Universal Robots PolyScope program: static_blocks.urp

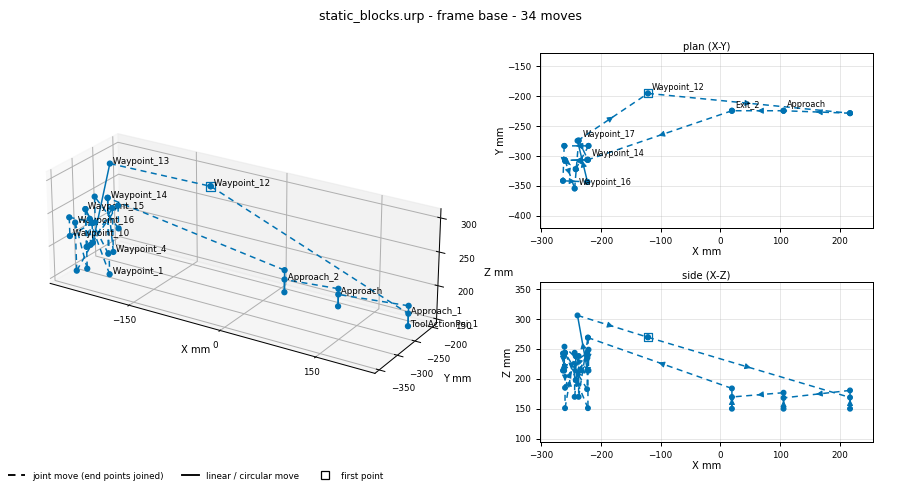
[picture p0: tool path of static_blocks.urp in frame base, 34 of 34 moves have a stored position in this frame; points joined in program order, loops and branches not executed]
Program static_blocks (installation=default directory=/programs/usbdisk createdIn=5.3.1.64192 lastSavedIn=5.3.1.64192 robotSerialNumber=20195300365)
Calibrated DH parameters: a=[-0.000093, -0.190649, -0.212673, 0.000091, -0.000205, 0]; d=[0.151591, 44.061648, -42.488068, -1.442789, 0.085322, 0.091911]; alpha=[1.570082, -0.003447, 0.007513, 1.572293, -1.571904, 0]; deltaTheta=[0, -0.672656, 0.728185, -0.055522, 0.000005, 0]
BeforeStart
  URCap Gripper Activate (Robotiq_Grippers, Robotiq Inc.) dataModel(ResetAndActivateKey=true)
  Wait Sleep waitTime=2
  URCap Gripper (Robotiq_Grippers, Robotiq Inc.) dataModel(position=50.0, force=100.0, speed=100.0, positionInDouble=50.0, forceInDouble=100.0, speedInDouble=100.0, slaveIds=[9], blocking=true)
Robot Program (runOnlyOnce=true)
  MoveJ speed 60 deg/s, acceleration 80 deg/s^2 (useActiveTCP=true) feature=Base
    Waypoint Waypoint_12: TCP in base x=-121.283 y=-195.081 z=269.514 mm, rx=-2.167 ry=2.2415 rz=-0.0076 rad; joints [-88.099, -64.133, -118.46, -88.049, 91.631, -85.899] deg
  next := "large_1"
  Loop Counting (count=11) loopVariable(name=Loop_1)
    'Block selection'
    If next ≟ "large_1"
      URCap Palletizing (pallet-impl, Universal Robots) dataModel(palletFeature=Base, isPalletizing=true, rememberTraversal=false, Length(key=objectHeight value=0.01 unit=M), Variable(key=layerNumberVariable, variable(name=Pallet_1_lno, initializeExpression=1)), Variable(key=layerCountingVariable, variable(name=Pallet_1_lct, initializeExpression=1)), Variable(key=handleSeparatorVariable, variable(name=Pallet_1_sep, initializeExpression=False)), Variable(key=totalCountVariable, variable(name=Pallet_1_tct, initializeExpression=1)), Variable(key=name, variable(name=Large_1)), Variable(key=referencePoint, variable(featureName=referencePoint)), Variable(key=separatorPoint, variable(featureName=separatorPoint)), Variable(key=globalCountingVariable, variable(name=Pallet_1_cnt1, initializeExpression=1))); state(isChildrenLocked=true)
        URCap Patterns (pallet-impl, Universal Robots) state(isChildrenLocked=true)
          URCap Pattern (pallet-impl, Universal Robots) dataModel(UUID=37575b9b-24e8-4b53-bf02-43d1c72f6588, patternType=LINE, objects=4, Variable(key=nameVariable, variable(name=Line_Pattern_1))); state(isChildrenLocked=true)
            URCap Item (pallet-impl, Universal Robots) dataModel(UUID=94ef26eb-0406-42c0-9c7a-a5d3f7661bb4, patternType=LINE, index=0, calibrationDeltaTheta=[3.1764833014445715E-7, -0.6726562497450229, 0.7281850965771859, -0.055521791881094344, 5.417975891638949E-6, -3.308891861480978E-7], calibrationA=[-9.327832644612732E-5, -0.19064944224513533, -0.21267280235524616, 9.135661128094068E-5, -2.046441875520248E-4, 0.0], calibrationD=[0.15159127566255157, 44.06164831948618, -42.48806757161077, -1.4427889341768174, 0.08532194966640622, 0.09191068481194639], calibrationAlpha=[1.5700823634315826, -0.0034467901999681192, 0.007512569451791506, 1.5722928534010268, -1.5719039470931155, 0.0], calibrationJointChecksum=[-1322437199, -1322307948, -1493592214, -1327938167, -1330538947, -1329494862], calibrationStatus=2, calibrationValidChecksum=true, baseToFeature=[0.0, 0.0, 0.0, 0.0, 0.0, 0.0], TCPOffset=[2.6818013665053098E-6, -8.523257610526525E-7, 3.187511623176098E-6, -5.221405753076122E-6, 1.0916503052633558E-5, 1.7823756412515186E-5], JointPositions(key=jointpositions, JointPosition(key=[1], Angle(key=pos value=-0.386285 unit=RAD)), JointPosition(key=[2], Angle(key=pos value=-1.772217 unit=RAD)), JointPosition(key=[3], Angle(key=pos value=-2.142066 unit=RAD)), JointPosition(key=[4], Angle(key=pos value=-0.803353 unit=RAD)), JointPosition(key=[5], Angle(key=pos value=1.570932 unit=RAD)), JointPosition(key=[6], Angle(key=pos value=-0.3815 unit=RAD))), Variable(key=variable, variable(name=StartItem_1)))
            URCap Item (pallet-impl, Universal Robots) dataModel(UUID=a723c821-374d-4fb7-a72e-4b4fba4af77d, patternType=LINE, index=1, calibrationDeltaTheta=[3.1764833014445715E-7, -0.6726562497450229, 0.7281850965771859, -0.055521791881094344, 5.417975891638949E-6, -3.308891861480978E-7], calibrationA=[-9.327832644612732E-5, -0.19064944224513533, -0.21267280235524616, 9.135661128094068E-5, -2.046441875520248E-4, 0.0], calibrationD=[0.15159127566255157, 44.06164831948618, -42.48806757161077, -1.4427889341768174, 0.08532194966640622, 0.09191068481194639], calibrationAlpha=[1.5700823634315826, -0.0034467901999681192, 0.007512569451791506, 1.5722928534010268, -1.5719039470931155, 0.0], calibrationJointChecksum=[-1322437199, -1322307948, -1493592214, -1327938167, -1330538947, -1329494862], calibrationStatus=2, calibrationValidChecksum=true, baseToFeature=[0.0, 0.0, 0.0, 0.0, 0.0, 0.0], TCPOffset=[-4.482752550050151E-6, -1.082257494983141E-5, -1.6687113393309971E-6, -3.080320700071801E-6, 2.847478995674553E-5, -7.719056088527975E-5], JointPositions(key=jointpositions, JointPosition(key=[1], Angle(key=pos value=-0.845813 unit=RAD)), JointPosition(key=[2], Angle(key=pos value=-2.443735 unit=RAD)), JointPosition(key=[3], Angle(key=pos value=-1.007946 unit=RAD)), JointPosition(key=[4], Angle(key=pos value=-1.263676 unit=RAD)), JointPosition(key=[5], Angle(key=pos value=1.569273 unit=RAD)), JointPosition(key=[6], Angle(key=pos value=-0.846194 unit=RAD))), Variable(key=variable, variable(name=EndItem_1)))
        URCap Layers (pallet-impl, Universal Robots) dataModel(separators=[false], selectedPatterns=[37575b9b-24e8-4b53-bf02-43d1c72f6588])
        URCap At Each Item (pallet-impl, Universal Robots) dataModel(selectedPattern=37575b9b-24e8-4b53-bf02-43d1c72f6588, selectedPosition=94ef26eb-0406-42c0-9c7a-a5d3f7661bb4, Approach_calibrationDeltaTheta=[3.1764833014445715E-7, -0.6726562497450229, 0.7281850965771859, -0.055521791881094344, 5.417975891638949E-6, -3.308891861480978E-7], Approach_calibrationA=[-9.327832644612732E-5, -0.19064944224513533, -0.21267280235524616, 9.135661128094068E-5, -2.046441875520248E-4, 0.0], Approach_calibrationD=[0.15159127566255157, 44.06164831948618, -42.48806757161077, -1.4427889341768174, 0.08532194966640622, 0.09191068481194639], Approach_calibrationAlpha=[1.5700823634315826, -0.0034467901999681192, 0.007512569451791506, 1.5722928534010268, -1.5719039470931155, 0.0], Approach_calibrationJointChecksum=[-1322437199, -1322307948, -1493592214, -1327938167, -1330538947, -1329494862], Approach_calibrationStatus=2, Approach_calibrationValidChecksum=true, Approach_baseToFeature=[0.0, 0.0, 0.0, 0.0, 0.0, 0.0], Approach_TCPOffset=[-1.4110221621399521E-6, -9.056105289340088E-6, -4.040316261583188E-6, -7.025378227736759E-6, 4.9770386753854616E-6, -2.713524910439085E-5], Exit_calibrationDeltaTheta=[3.1764833014445715E-7, -0.6726562497450229, 0.7281850965771859, -0.055521791881094344, 5.417975891638949E-6, -3.308891861480978E-7], Exit_calibrationA=[-9.327832644612732E-5, -0.19064944224513533, -0.21267280235524616, 9.135661128094068E-5, -2.046441875520248E-4, 0.0], Exit_calibrationD=[0.15159127566255157, 44.06164831948618, -42.48806757161077, -1.4427889341768174, 0.08532194966640622, 0.09191068481194639], Exit_calibrationAlpha=[1.5700823634315826, -0.0034467901999681192, 0.007512569451791506, 1.5722928534010268, -1.5719039470931155, 0.0], Exit_calibrationJointChecksum=[-1322437199, -1322307948, -1493592214, -1327938167, -1330538947, -1329494862], Exit_calibrationStatus=2, Exit_calibrationValidChecksum=true, Exit_baseToFeature=[0.0, 0.0, 0.0, 0.0, 0.0, 0.0], Exit_TCPOffset=[4.440688230411549E-6, 1.0608106728315914E-5, 6.984684250199713E-6, -3.32523645938351E-5, 8.927854697233474E-6, -3.551786211011088E-5], currentWizardState=LANDING, Pose(key=refBaseToFeature, Position(key=posePosition, Length(key=X value=0 unit=M), Length(key=Y value=0 unit=M), Length(key=Z value=0 unit=M)), Rotation(key=poseRotation, Angle(key=RX value=0 unit=RAD), Angle(key=RY value=0 unit=RAD), Angle(key=RZ value=0 unit=RAD))), Pose(key=refPose, Position(key=posePosition, Length(key=X value=0.216857 unit=M), Length(key=Y value=-0.228211 unit=M), Length(key=Z value=0.149941 unit=M)), Rotation(key=poseRotation, Angle(key=RX value=2.221569 unit=RAD), Angle(key=RY value=-2.213073 unit=RAD), Angle(key=RZ value=-0.006933 unit=RAD))), JointPositions(key=Approach_jointpositions, JointPosition(key=[1], Angle(key=pos value=-0.386188 unit=RAD)), JointPosition(key=[2], Angle(key=pos value=-1.712734 unit=RAD)), JointPosition(key=[3], Angle(key=pos value=-2.099671 unit=RAD)), JointPosition(key=[4], Angle(key=pos value=-0.90523 unit=RAD)), JointPosition(key=[5], Angle(key=pos value=1.571526 unit=RAD)), JointPosition(key=[6], Angle(key=pos value=-0.381836 unit=RAD))), JointPositions(key=Exit_jointpositions, JointPosition(key=[1], Angle(key=pos value=-0.386112 unit=RAD)), JointPosition(key=[2], Angle(key=pos value=-1.679803 unit=RAD)), JointPosition(key=[3], Angle(key=pos value=-2.069692 unit=RAD)), JointPosition(key=[4], Angle(key=pos value=-0.968137 unit=RAD)), JointPosition(key=[5], Angle(key=pos value=1.571865 unit=RAD)), JointPosition(key=[6], Angle(key=pos value=-0.382075 unit=RAD))))
          URCap Generated Movements (pallet-impl, Universal Robots) state(isChildrenLocked=true)
            MoveJ speed 60 deg/s, acceleration 80 deg/s^2 (useActiveTCP=true) feature=referencePoint
              Waypoint Approach_1: TCP in base x=216.866 y=-228.21 z=168.787 mm, rx=2.2216 ry=-2.213 rz=-0.0069 rad; joints [-22.126, -98.133, -120.3, -51.868, 90.041, -21.878] deg; TCP offset x=0 y=0 z=0 mm, rx=0 ry=0 rz=0 rad; feature pose in base x=216.857 y=-228.211 z=149.941 mm, rx=2.2216 ry=-2.2131 rz=-0.0069 rad
            MoveL speed 250 mm/s, acceleration 1200 mm/s^2 (useActiveTCP=true) feature(featureName=referencePoint)
              Waypoint ToolActionPoi_1: TCP in base x=216.857 y=-228.211 z=149.941 mm, rx=2.2216 ry=-2.2131 rz=-0.0069 rad; joints [-22.133, -101.542, -122.731, -46.028, 90.007, -21.858] deg; TCP offset x=0 y=0 z=0 mm, rx=0 ry=0 rz=0 rad
            Folder Tool action
              URCap Gripper (Robotiq_Grippers, Robotiq Inc.) dataModel(position=100.0, force=100.0, speed=100.0, positionInDouble=100.0, forceInDouble=100.0, speedInDouble=100.0, slaveIds=[9], blocking=true)
            MoveL speed 250 mm/s, acceleration 1200 mm/s^2 (useActiveTCP=true) feature(featureName=referencePoint)
              Waypoint Exit_1: motionParameters(blendRadius=0.015); TCP in base x=216.847 y=-228.216 z=180.576 mm, rx=2.2216 ry=-2.213 rz=-0.007 rad; joints [-22.124, -96.246, -118.586, -55.47, 90.06, -21.895] deg; TCP offset x=0 y=0 z=0 mm, rx=0 ry=0 rz=0 rad
    ElseIf next ≟ "small_1"
      URCap Palletizing (pallet-impl, Universal Robots) dataModel(palletFeature=Base, isPalletizing=true, rememberTraversal=false, Length(key=objectHeight value=0.01 unit=M), Variable(key=layerNumberVariable, variable(name=Pallet_1_lno_1, initializeExpression=1)), Variable(key=layerCountingVariable, variable(name=Pallet_1_lct_1, initializeExpression=1)), Variable(key=handleSeparatorVariable, variable(name=Pallet_1_sep_1, initializeExpression=False)), Variable(key=totalCountVariable, variable(name=Pallet_1_tct_1, initializeExpression=1)), Variable(key=name, variable(name=Small_1)), Variable(key=referencePoint, variable(featureName=referencePoin_1)), Variable(key=separatorPoint, variable(featureName=separatorPoin_1)), Variable(key=globalCountingVariable, variable(name=Pallet_1_cnt2, initializeExpression=1))); state(isChildrenLocked=true)
        URCap Patterns (pallet-impl, Universal Robots) state(isChildrenLocked=true)
          URCap Pattern (pallet-impl, Universal Robots) dataModel(UUID=8f5fe08d-2c45-49f2-8f1a-65c607567d74, patternType=LINE, objects=4, Variable(key=nameVariable, variable(name=Line_Pattern_2))); state(isChildrenLocked=true)
            URCap Item (pallet-impl, Universal Robots) dataModel(UUID=ef528854-cb52-475c-81ed-63f5d340cd60, patternType=LINE, index=0, calibrationDeltaTheta=[3.1764833014445715E-7, -0.6726562497450229, 0.7281850965771859, -0.055521791881094344, 5.417975891638949E-6, -3.308891861480978E-7], calibrationA=[-9.327832644612732E-5, -0.19064944224513533, -0.21267280235524616, 9.135661128094068E-5, -2.046441875520248E-4, 0.0], calibrationD=[0.15159127566255157, 44.06164831948618, -42.48806757161077, -1.4427889341768174, 0.08532194966640622, 0.09191068481194639], calibrationAlpha=[1.5700823634315826, -0.0034467901999681192, 0.007512569451791506, 1.5722928534010268, -1.5719039470931155, 0.0], calibrationJointChecksum=[-1322437199, -1322307948, -1493592214, -1327938167, -1330538947, -1329494862], calibrationStatus=2, calibrationValidChecksum=true, baseToFeature=[0.0, 0.0, 0.0, 0.0, 0.0, 0.0], TCPOffset=[7.196090374694819E-7, -7.525119034013095E-7, 2.3613486090923175E-6, -5.861788620822338E-6, -1.7185264349297415E-5, 1.0867011174151283E-5], JointPositions(key=jointpositions, JointPosition(key=[1], Angle(key=pos value=-0.579147 unit=RAD)), JointPosition(key=[2], Angle(key=pos value=-1.475214 unit=RAD)), JointPosition(key=[3], Angle(key=pos value=-2.46543 unit=RAD)), JointPosition(key=[4], Angle(key=pos value=-0.776185 unit=RAD)), JointPosition(key=[5], Angle(key=pos value=1.570404 unit=RAD)), JointPosition(key=[6], Angle(key=pos value=-0.573518 unit=RAD))), Variable(key=variable, variable(name=StartItem_2)))
            URCap Item (pallet-impl, Universal Robots) dataModel(UUID=c15b3bae-27b4-4f22-a9be-ccead8772f48, patternType=LINE, index=1, calibrationDeltaTheta=[3.1764833014445715E-7, -0.6726562497450229, 0.7281850965771859, -0.055521791881094344, 5.417975891638949E-6, -3.308891861480978E-7], calibrationA=[-9.327832644612732E-5, -0.19064944224513533, -0.21267280235524616, 9.135661128094068E-5, -2.046441875520248E-4, 0.0], calibrationD=[0.15159127566255157, 44.06164831948618, -42.48806757161077, -1.4427889341768174, 0.08532194966640622, 0.09191068481194639], calibrationAlpha=[1.5700823634315826, -0.0034467901999681192, 0.007512569451791506, 1.5722928534010268, -1.5719039470931155, 0.0], calibrationJointChecksum=[-1322437199, -1322307948, -1493592214, -1327938167, -1330538947, -1329494862], calibrationStatus=2, calibrationValidChecksum=true, baseToFeature=[0.0, 0.0, 0.0, 0.0, 0.0, 0.0], TCPOffset=[6.867596638648887E-6, 1.6127585317354809E-6, -1.4517486032261662E-5, -5.9295253787075885E-6, 7.61064027945187E-5, -1.3647353319639889E-5], JointPositions(key=jointpositions, JointPosition(key=[1], Angle(key=pos value=-1.056839 unit=RAD)), JointPosition(key=[2], Angle(key=pos value=-2.273802 unit=RAD)), JointPosition(key=[3], Angle(key=pos value=-1.326947 unit=RAD)), JointPosition(key=[4], Angle(key=pos value=-1.113261 unit=RAD)), JointPosition(key=[5], Angle(key=pos value=1.568262 unit=RAD)), JointPosition(key=[6], Angle(key=pos value=-1.055578 unit=RAD))), Variable(key=variable, variable(name=EndItem_2)))
        URCap Layers (pallet-impl, Universal Robots) dataModel(separators=[false], selectedPatterns=[8f5fe08d-2c45-49f2-8f1a-65c607567d74])
        URCap At Each Item (pallet-impl, Universal Robots) dataModel(selectedPattern=8f5fe08d-2c45-49f2-8f1a-65c607567d74, selectedPosition=ef528854-cb52-475c-81ed-63f5d340cd60, Approach_calibrationDeltaTheta=[3.1764833014445715E-7, -0.6726562497450229, 0.7281850965771859, -0.055521791881094344, 5.417975891638949E-6, -3.308891861480978E-7], Approach_calibrationA=[-9.327832644612732E-5, -0.19064944224513533, -0.21267280235524616, 9.135661128094068E-5, -2.046441875520248E-4, 0.0], Approach_calibrationD=[0.15159127566255157, 44.06164831948618, -42.48806757161077, -1.4427889341768174, 0.08532194966640622, 0.09191068481194639], Approach_calibrationAlpha=[1.5700823634315826, -0.0034467901999681192, 0.007512569451791506, 1.5722928534010268, -1.5719039470931155, 0.0], Approach_calibrationJointChecksum=[-1322437199, -1322307948, -1493592214, -1327938167, -1330538947, -1329494862], Approach_calibrationStatus=2, Approach_calibrationValidChecksum=true, Approach_baseToFeature=[0.0, 0.0, 0.0, 0.0, 0.0, 0.0], Approach_TCPOffset=[-1.8296166631182054E-6, -5.2785861738846585E-6, 4.523678061779668E-6, -2.6542376188082585E-5, -8.975232779585173E-6, -3.1784731117598936E-5], Exit_calibrationDeltaTheta=[3.1764833014445715E-7, -0.6726562497450229, 0.7281850965771859, -0.055521791881094344, 5.417975891638949E-6, -3.308891861480978E-7], Exit_calibrationA=[-9.327832644612732E-5, -0.19064944224513533, -0.21267280235524616, 9.135661128094068E-5, -2.046441875520248E-4, 0.0], Exit_calibrationD=[0.15159127566255157, 44.06164831948618, -42.48806757161077, -1.4427889341768174, 0.08532194966640622, 0.09191068481194639], Exit_calibrationAlpha=[1.5700823634315826, -0.0034467901999681192, 0.007512569451791506, 1.5722928534010268, -1.5719039470931155, 0.0], Exit_calibrationJointChecksum=[-1322437199, -1322307948, -1493592214, -1327938167, -1330538947, -1329494862], Exit_calibrationStatus=2, Exit_calibrationValidChecksum=true, Exit_baseToFeature=[0.0, 0.0, 0.0, 0.0, 0.0, 0.0], Exit_TCPOffset=[-1.517237854353759E-6, -9.613929180279923E-6, -6.434422402695761E-6, 9.261849516252882E-6, 1.6687881217173567E-5, -3.51484445230019E-5], currentWizardState=LANDING, Pose(key=refBaseToFeature, Position(key=posePosition, Length(key=X value=0 unit=M), Length(key=Y value=0 unit=M), Length(key=Z value=0 unit=M)), Rotation(key=poseRotation, Angle(key=RX value=0 unit=RAD), Angle(key=RY value=0 unit=RAD), Angle(key=RZ value=0 unit=RAD))), Pose(key=refPose, Position(key=posePosition, Length(key=X value=0.105616 unit=M), Length(key=Y value=-0.224089 unit=M), Length(key=Z value=0.149939 unit=M)), Rotation(key=poseRotation, Angle(key=RX value=2.221562 unit=RAD), Angle(key=RY value=-2.213091 unit=RAD), Angle(key=RZ value=-0.006958 unit=RAD))), JointPositions(key=Approach_jointpositions, JointPosition(key=[1], Angle(key=pos value=-0.578996 unit=RAD)), JointPosition(key=[2], Angle(key=pos value=-1.398829 unit=RAD)), JointPosition(key=[3], Angle(key=pos value=-2.412 unit=RAD)), JointPosition(key=[4], Angle(key=pos value=-0.906009 unit=RAD)), JointPosition(key=[5], Angle(key=pos value=1.571251 unit=RAD)), JointPosition(key=[6], Angle(key=pos value=-0.573984 unit=RAD))), JointPositions(key=Exit_jointpositions, JointPosition(key=[1], Angle(key=pos value=-0.578911 unit=RAD)), JointPosition(key=[2], Angle(key=pos value=-1.367711 unit=RAD)), JointPosition(key=[3], Angle(key=pos value=-2.384276 unit=RAD)), JointPosition(key=[4], Angle(key=pos value=-0.96485 unit=RAD)), JointPosition(key=[5], Angle(key=pos value=1.571588 unit=RAD)), JointPosition(key=[6], Angle(key=pos value=-0.574219 unit=RAD))))
          URCap Generated Movements (pallet-impl, Universal Robots) state(isChildrenLocked=true)
            MoveJ speed 60 deg/s, acceleration 80 deg/s^2 (useActiveTCP=true) feature=referencePoin_1
              Waypoint Approach: TCP in base x=105.622 y=-224.087 z=168.076 mm, rx=2.2216 ry=-2.213 rz=-0.007 rad; joints [-33.173, -80.148, -138.197, -51.911, 90.026, -32.887] deg; TCP offset x=0 y=0 z=0 mm, rx=0 ry=0 rz=0 rad; feature pose in base x=105.616 y=-224.089 z=149.939 mm, rx=2.2216 ry=-2.2131 rz=-0.007 rad
            MoveL speed 250 mm/s, acceleration 1200 mm/s^2 (useActiveTCP=true) feature(featureName=referencePoin_1)
              Waypoint ToolActionPoint: TCP in base x=105.616 y=-224.089 z=149.939 mm, rx=2.2216 ry=-2.2131 rz=-0.007 rad; joints [-33.183, -84.525, -141.258, -44.472, 89.978, -32.86] deg; TCP offset x=0 y=0 z=0 mm, rx=0 ry=0 rz=0 rad
            Folder Tool action
              URCap Gripper (Robotiq_Grippers, Robotiq Inc.) dataModel(position=100.0, force=100.0, speed=100.0, positionInDouble=100.0, forceInDouble=100.0, speedInDouble=100.0, slaveIds=[9], blocking=true)
            MoveL speed 250 mm/s, acceleration 1200 mm/s^2 (useActiveTCP=true) feature(featureName=referencePoin_1)
              Waypoint Exit: motionParameters(blendRadius=0.015); TCP in base x=105.626 y=-224.087 z=176.77 mm, rx=2.2216 ry=-2.213 rz=-0.0069 rad; joints [-33.167, -78.363, -136.608, -55.283, 90.045, -32.9] deg; TCP offset x=0 y=0 z=0 mm, rx=0 ry=0 rz=0 rad
    Else 
      URCap Palletizing (pallet-impl, Universal Robots) dataModel(palletFeature=Base, isPalletizing=true, rememberTraversal=false, Length(key=objectHeight value=0.01 unit=M), Variable(key=layerNumberVariable, variable(name=Pallet_3_lno, initializeExpression=1)), Variable(key=layerCountingVariable, variable(name=Pallet_3_lct, initializeExpression=1)), Variable(key=handleSeparatorVariable, variable(name=Pallet_3_sep, initializeExpression=False)), Variable(key=totalCountVariable, variable(name=Pallet_3_tct, initializeExpression=1)), Variable(key=name, variable(name=Small_2)), Variable(key=referencePoint, variable(featureName=referencePoin_2)), Variable(key=separatorPoint, variable(featureName=separatorPoin_2)), Variable(key=globalCountingVariable, variable(name=Pallet_3_cnt1, initializeExpression=1))); state(isChildrenLocked=true)
        URCap Patterns (pallet-impl, Universal Robots) state(isChildrenLocked=true)
          URCap Pattern (pallet-impl, Universal Robots) dataModel(UUID=574e648a-9869-4bcb-a6fe-864b98b65979, patternType=LINE, objects=4, Variable(key=nameVariable, variable(name=Line_Pattern_3))); state(isChildrenLocked=true)
            URCap Item (pallet-impl, Universal Robots) dataModel(UUID=3619f09d-97e3-4d4e-aeec-a5329e7c8f8b, patternType=LINE, index=0, calibrationDeltaTheta=[3.1764833014445715E-7, -0.6726562497450229, 0.7281850965771859, -0.055521791881094344, 5.417975891638949E-6, -3.308891861480978E-7], calibrationA=[-9.327832644612732E-5, -0.19064944224513533, -0.21267280235524616, 9.135661128094068E-5, -2.046441875520248E-4, 0.0], calibrationD=[0.15159127566255157, 44.06164831948618, -42.48806757161077, -1.4427889341768174, 0.08532194966640622, 0.09191068481194639], calibrationAlpha=[1.5700823634315826, -0.0034467901999681192, 0.007512569451791506, 1.5722928534010268, -1.5719039470931155, 0.0], calibrationJointChecksum=[-1322437199, -1322307948, -1493592214, -1327938167, -1330538947, -1329494862], calibrationStatus=2, calibrationValidChecksum=true, baseToFeature=[0.0, 0.0, 0.0, 0.0, 0.0, 0.0], TCPOffset=[-1.471914889417114E-7, -9.062111944835999E-6, 4.858574105065516E-6, -6.559488045899108E-6, -1.3766923162685491E-5, -5.608483778319356E-6], JointPositions(key=jointpositions, JointPosition(key=[1], Angle(key=pos value=-0.869663 unit=RAD)), JointPosition(key=[2], Angle(key=pos value=-1.338984 unit=RAD)), JointPosition(key=[3], Angle(key=pos value=-2.567281 unit=RAD)), JointPosition(key=[4], Angle(key=pos value=-0.808969 unit=RAD)), JointPosition(key=[5], Angle(key=pos value=1.569596 unit=RAD)), JointPosition(key=[6], Angle(key=pos value=-0.863997 unit=RAD))), Variable(key=variable, variable(name=StartItem_3)))
            URCap Item (pallet-impl, Universal Robots) dataModel(UUID=43353e96-12ed-4b99-95b5-f18523ae2f1f, patternType=LINE, index=1, calibrationDeltaTheta=[3.1764833014445715E-7, -0.6726562497450229, 0.7281850965771859, -0.055521791881094344, 5.417975891638949E-6, -3.308891861480978E-7], calibrationA=[-9.327832644612732E-5, -0.19064944224513533, -0.21267280235524616, 9.135661128094068E-5, -2.046441875520248E-4, 0.0], calibrationD=[0.15159127566255157, 44.06164831948618, -42.48806757161077, -1.4427889341768174, 0.08532194966640622, 0.09191068481194639], calibrationAlpha=[1.5700823634315826, -0.0034467901999681192, 0.007512569451791506, 1.5722928534010268, -1.5719039470931155, 0.0], calibrationJointChecksum=[-1322437199, -1322307948, -1493592214, -1327938167, -1330538947, -1329494862], calibrationStatus=2, calibrationValidChecksum=true, baseToFeature=[0.0, 0.0, 0.0, 0.0, 0.0, 0.0], TCPOffset=[-2.699244438297832E-6, -1.993162529571879E-7, -2.2601341719635792E-5, 2.6517761326188484E-5, 3.333393093251858E-5, 1.450252224784447E-5], JointPositions(key=jointpositions, JointPosition(key=[1], Angle(key=pos value=-1.246701 unit=RAD)), JointPosition(key=[2], Angle(key=pos value=-2.204283 unit=RAD)), JointPosition(key=[3], Angle(key=pos value=-1.452761 unit=RAD)), JointPosition(key=[4], Angle(key=pos value=-1.055644 unit=RAD)), JointPosition(key=[5], Angle(key=pos value=1.567749 unit=RAD)), JointPosition(key=[6], Angle(key=pos value=-1.24482 unit=RAD))), Variable(key=variable, variable(name=EndItem_3)))
        URCap Layers (pallet-impl, Universal Robots) dataModel(separators=[false], selectedPatterns=[574e648a-9869-4bcb-a6fe-864b98b65979])
        URCap At Each Item (pallet-impl, Universal Robots) dataModel(selectedPattern=574e648a-9869-4bcb-a6fe-864b98b65979, selectedPosition=3619f09d-97e3-4d4e-aeec-a5329e7c8f8b, Approach_calibrationDeltaTheta=[3.1764833014445715E-7, -0.6726562497450229, 0.7281850965771859, -0.055521791881094344, 5.417975891638949E-6, -3.308891861480978E-7], Approach_calibrationA=[-9.327832644612732E-5, -0.19064944224513533, -0.21267280235524616, 9.135661128094068E-5, -2.046441875520248E-4, 0.0], Approach_calibrationD=[0.15159127566255157, 44.06164831948618, -42.48806757161077, -1.4427889341768174, 0.08532194966640622, 0.09191068481194639], Approach_calibrationAlpha=[1.5700823634315826, -0.0034467901999681192, 0.007512569451791506, 1.5722928534010268, -1.5719039470931155, 0.0], Approach_calibrationJointChecksum=[-1322437199, -1322307948, -1493592214, -1327938167, -1330538947, -1329494862], Approach_calibrationStatus=2, Approach_calibrationValidChecksum=true, Approach_baseToFeature=[0.0, 0.0, 0.0, 0.0, 0.0, 0.0], Approach_TCPOffset=[1.7216837140676677E-6, -3.506743741481938E-6, -1.0808390142336144E-6, -1.6443935207651089E-6, 4.86080167331034E-6, -2.9982690882012256E-5], Exit_calibrationDeltaTheta=[3.1764833014445715E-7, -0.6726562497450229, 0.7281850965771859, -0.055521791881094344, 5.417975891638949E-6, -3.308891861480978E-7], Exit_calibrationA=[-9.327832644612732E-5, -0.19064944224513533, -0.21267280235524616, 9.135661128094068E-5, -2.046441875520248E-4, 0.0], Exit_calibrationD=[0.15159127566255157, 44.06164831948618, -42.48806757161077, -1.4427889341768174, 0.08532194966640622, 0.09191068481194639], Exit_calibrationAlpha=[1.5700823634315826, -0.0034467901999681192, 0.007512569451791506, 1.5722928534010268, -1.5719039470931155, 0.0], Exit_calibrationJointChecksum=[-1322437199, -1322307948, -1493592214, -1327938167, -1330538947, -1329494862], Exit_calibrationStatus=2, Exit_calibrationValidChecksum=true, Exit_baseToFeature=[0.0, 0.0, 0.0, 0.0, 0.0, 0.0], Exit_TCPOffset=[-4.7682124618142474E-7, -1.929772925179929E-6, -1.986456084873689E-6, 4.125717686270397E-6, -2.831162655691365E-6, 4.997597875419577E-8], currentWizardState=LANDING, Pose(key=refBaseToFeature, Position(key=posePosition, Length(key=X value=0 unit=M), Length(key=Y value=0 unit=M), Length(key=Z value=0 unit=M)), Rotation(key=poseRotation, Angle(key=RX value=0 unit=RAD), Angle(key=RY value=0 unit=RAD), Angle(key=RZ value=0 unit=RAD))), Pose(key=refPose, Position(key=posePosition, Length(key=X value=0.019209 unit=M), Length(key=Y value=-0.224088 unit=M), Length(key=Z value=0.149936 unit=M)), Rotation(key=poseRotation, Angle(key=RX value=2.221578 unit=RAD), Angle(key=RY value=-2.213071 unit=RAD), Angle(key=RZ value=-0.006955 unit=RAD))), JointPositions(key=Approach_jointpositions, JointPosition(key=[1], Angle(key=pos value=-0.869398 unit=RAD)), JointPosition(key=[2], Angle(key=pos value=-1.250368 unit=RAD)), JointPosition(key=[3], Angle(key=pos value=-2.50146 unit=RAD)), JointPosition(key=[4], Angle(key=pos value=-0.963415 unit=RAD)), JointPosition(key=[5], Angle(key=pos value=1.570564 unit=RAD)), JointPosition(key=[6], Angle(key=pos value=-0.864557 unit=RAD))), JointPositions(key=Exit_jointpositions, JointPosition(key=[1], Angle(key=pos value=-0.869215 unit=RAD)), JointPosition(key=[2], Angle(key=pos value=-1.200405 unit=RAD)), JointPosition(key=[3], Angle(key=pos value=-2.449496 unit=RAD)), JointPosition(key=[4], Angle(key=pos value=-1.065339 unit=RAD)), JointPosition(key=[5], Angle(key=pos value=1.571095 unit=RAD)), JointPosition(key=[6], Angle(key=pos value=-0.86499 unit=RAD))))
          URCap Generated Movements (pallet-impl, Universal Robots) state(isChildrenLocked=true)
            MoveJ speed 60 deg/s, acceleration 80 deg/s^2 (useActiveTCP=true) feature=referencePoin_2
              Waypoint Approach_2: TCP in base x=19.213 y=-224.089 z=169.579 mm, rx=2.2216 ry=-2.213 rz=-0.007 rad; joints [-49.812, -71.641, -143.323, -55.2, 89.986, -49.537] deg; TCP offset x=0 y=0 z=0 mm, rx=0 ry=0 rz=0 rad; feature pose in base x=19.209 y=-224.088 z=149.936 mm, rx=2.2216 ry=-2.2131 rz=-0.007 rad
            MoveL speed 250 mm/s, acceleration 1200 mm/s^2 (useActiveTCP=true) feature(featureName=referencePoin_2)
              Waypoint ToolActionPoi_2: TCP in base x=19.209 y=-224.088 z=149.936 mm, rx=2.2216 ry=-2.2131 rz=-0.007 rad; joints [-49.826, -76.72, -147.095, -46.349, 89.931, -49.502] deg; TCP offset x=0 y=0 z=0 mm, rx=0 ry=0 rz=0 rad
            Folder Tool action
              URCap Gripper (Robotiq_Grippers, Robotiq Inc.) dataModel(position=100.0, force=100.0, speed=100.0, positionInDouble=100.0, forceInDouble=100.0, speedInDouble=100.0, slaveIds=[9], blocking=true)
            MoveL speed 250 mm/s, acceleration 1200 mm/s^2 (useActiveTCP=true) feature(featureName=referencePoin_2)
              Waypoint Exit_2: motionParameters(blendRadius=0.015); TCP in base x=19.211 y=-224.087 z=183.922 mm, rx=2.2216 ry=-2.2131 rz=-0.007 rad; joints [-49.802, -68.778, -140.345, -61.04, 90.017, -49.56] deg; TCP offset x=0 y=0 z=0 mm, rx=0 ry=0 rz=0 rad
    'Build Movement based on loop count'
    Switch expression=Loop_1
      Case (caseValue=0)
        MoveJ speed 80 deg/s, acceleration 80 deg/s^2 (useActiveTCP=true) feature=Base
          Waypoint Waypoint_14: motionParameters(blendRadius=0.025); TCP in base x=-221.702 y=-306.123 z=268.895 mm, rx=3.071 ry=-0.0057 rz=-0.0036 rad; joints [-106.085, -102.763, -86.83, -76.411, 91.286, -195.56] deg
          Waypoint Waypoint_1: TCP in base x=-221.711 y=-306.113 z=150.84 mm, rx=3.071 ry=-0.0058 rz=-0.0036 rad; joints [-106.136, -114.449, -105.748, -45.809, 91.172, -195.438] deg
        next := "large_1"
      Case (caseValue=1)
        MoveJ speed 80 deg/s, acceleration 80 deg/s^2 (useActiveTCP=true) feature=Base
          Waypoint Waypoint_15: motionParameters(blendRadius=0.025); TCP in base x=-260.029 y=-307.245 z=243.485 mm, rx=3.071 ry=-0.0058 rz=-0.0035 rad; joints [-111.758, -110.064, -84.044, -72.013, 91.65, -201.204] deg
          Waypoint Waypoint_2: TCP in base x=-260.023 y=-307.26 z=150.834 mm, rx=3.071 ry=-0.0058 rz=-0.0036 rad; joints [-111.789, -119.387, -97.491, -49.242, 91.562, -201.114] deg
        next := "small_1"
      Case (caseValue=2)
        MoveJ speed 80 deg/s, acceleration 80 deg/s^2 (useActiveTCP=true) feature=Base
          Waypoint Waypoint_16: motionParameters(blendRadius=0.025); TCP in base x=-243.935 y=-354.168 z=243.603 mm, rx=2.1533 ry=-2.2814 rz=0.0711 rad; joints [-107.442, -117.648, -71.84, -78.991, 92.448, -103.884] deg
          Waypoint Waypoint_3: TCP in base x=-243.953 y=-354.156 z=169.839 mm, rx=2.1533 ry=-2.2815 rz=0.071 rad; joints [-107.476, -123.165, -83.897, -61.417, 92.404, -103.807] deg
        next := "small_1"
      Case (caseValue=3)
        MoveJ speed 80 deg/s, acceleration 80 deg/s^2 (useActiveTCP=true) feature=Base
          Waypoint Waypoint_17: motionParameters(blendRadius=0.025); TCP in base x=-237.256 y=-273.962 z=238.187 mm, rx=2.1533 ry=-2.2814 rz=0.071 rad; joints [-110.535, -101.491, -95.81, -71.293, 92.537, -106.872] deg
          Waypoint Waypoint_4: TCP in base x=-237.256 y=-273.956 z=169.84 mm, rx=2.1533 ry=-2.2814 rz=0.071 rad; joints [-110.564, -108.719, -106.727, -53.146, 92.466, -106.798] deg
        next := "large_1"
      Case (caseValue=4)
        MoveJ speed 80 deg/s, acceleration 80 deg/s^2 (useActiveTCP=true) feature=Base
          Waypoint Waypoint_14: motionParameters(blendRadius=0.025); TCP in base x=-221.702 y=-306.123 z=268.895 mm, rx=3.071 ry=-0.0057 rz=-0.0036 rad; joints [-106.085, -102.763, -86.83, -76.411, 91.286, -195.56] deg
          Waypoint Waypoint_5: TCP in base x=-223.118 y=-306.108 z=182.707 mm, rx=3.071 ry=-0.0057 rz=-0.0036 rad; joints [-106.349, -110.107, -101.836, -54.069, 91.23, -195.688] deg
        next := "large_1"
      Case (caseValue=5)
        MoveJ speed 80 deg/s, acceleration 80 deg/s^2 (useActiveTCP=true) feature=Base
          Waypoint Waypoint_15: motionParameters(blendRadius=0.025); TCP in base x=-260.029 y=-307.245 z=243.485 mm, rx=3.071 ry=-0.0058 rz=-0.0035 rad; joints [-111.758, -110.064, -84.044, -72.013, 91.65, -201.204] deg
          Waypoint Waypoint_6: TCP in base x=-260.029 y=-307.259 z=185.017 mm, rx=3.071 ry=-0.0058 rz=-0.0036 rad; joints [-111.781, -115.041, -93.624, -57.455, 91.6, -201.142] deg
        next := "small_1"
      Case (caseValue=6)
        MoveJ speed 80 deg/s, acceleration 80 deg/s^2 (useActiveTCP=true) feature=Base
          Waypoint Waypoint_18: motionParameters(blendRadius=0.025); TCP in base x=-242.146 y=-321.909 z=237.971 mm, rx=-2.1081 ry=2.2853 rz=-0.0296 rad; joints [-108.583, -111.86, -80.951, -78.217, 92.143, -103.73] deg
          Waypoint Waypoint_7: TCP in base x=-242.149 y=-321.9 z=197.927 mm, rx=-2.1081 ry=2.2853 rz=-0.0296 rad; joints [-108.603, -114.722, -88.04, -68.266, 92.12, -103.686] deg
        next := "small_1"
      Case (caseValue=7)
        MoveJ speed 80 deg/s, acceleration 80 deg/s^2 (useActiveTCP=true) feature=Base
          Waypoint Waypoint_19: motionParameters(blendRadius=0.025); TCP in base x=-220.731 y=-282.828 z=248.802 mm, rx=3.1163 ry=-0.0886 rz=-0.012 rad; joints [-106.762, -99.566, -95.207, -73.722, 90.244, -193.192] deg
          Waypoint Waypoint_8: TCP in base x=-220.729 y=-282.826 z=213.758 mm, rx=3.1163 ry=-0.0886 rz=-0.012 rad; joints [-106.78, -102.314, -101.819, -64.362, 90.217, -193.151] deg
        next := "small_2"
      Case (caseValue=8)
        MoveJ speed 80 deg/s, acceleration 80 deg/s^2 (useActiveTCP=true) feature=Base
          Waypoint Waypoint_20: motionParameters(blendRadius=0.025); TCP in base x=-260.991 y=-282.899 z=253.768 mm, rx=3.1161 ry=-0.0885 rz=-0.012 rad; joints [-113.008, -105.708, -86.112, -76.666, 90.395, -199.478] deg
          Waypoint Waypoint_9: TCP in base x=-261.455 y=-282.841 z=213.804 mm, rx=3.1161 ry=-0.0885 rz=-0.012 rad; joints [-113.1, -108.485, -93.596, -66.405, 90.371, -199.505] deg
        next := "small_2"
      Case (caseValue=9)
        MoveJ speed 80 deg/s, acceleration 80 deg/s^2 (useActiveTCP=true) feature=Base
          Waypoint Waypoint_21: motionParameters(blendRadius=0.025); TCP in base x=-263.496 y=-341.337 z=242.416 mm, rx=3.1162 ry=-0.0886 rz=-0.0118 rad; joints [-110.122, -117.729, -72.015, -78.743, 90.311, -196.642] deg
          Waypoint Waypoint_10: TCP in base x=-263.489 y=-341.336 z=213.776 mm, rx=3.1162 ry=-0.0886 rz=-0.0118 rad; joints [-110.136, -119.309, -77.46, -71.719, 90.299, -196.612] deg
        next := "small_2"
      Case (caseValue=10)
        MoveJ speed 80 deg/s, acceleration 80 deg/s^2 (useActiveTCP=true) feature=Base
          Waypoint Waypoint_22: motionParameters(blendRadius=0.025); TCP in base x=-222.892 y=-343.041 z=243.423 mm, rx=3.1162 ry=-0.0886 rz=-0.0121 rad; joints [-104.472, -112.124, -80.098, -76.27, 90.164, -190.959] deg
          Waypoint Waypoint_11: TCP in base x=-222.547 y=-343.002 z=213.787 mm, rx=3.1162 ry=-0.0886 rz=-0.0121 rad; joints [-104.439, -113.979, -85.666, -68.847, 90.145, -190.877] deg
        next := ""
    URCap Gripper (Robotiq_Grippers, Robotiq Inc.) dataModel(position=50.0, force=100.0, speed=100.0, positionInDouble=50.0, forceInDouble=100.0, speedInDouble=100.0, slaveIds=[9], blocking=true)
    MoveL speed 400 mm/s, acceleration 1200 mm/s^2 (useActiveTCP=true) feature=Base
      Waypoint Waypoint_13: motionParameters(blendRadius=0.05); TCP in base x=-239.189 y=-274.297 z=306.068 mm, rx=-2.1503 ry=2.2577 rz=0.0063 rad; joints [-110.266, -100.403, -77.534, -93.321, 90.715, -107.307] deg
  MoveJ speed 60 deg/s, acceleration 80 deg/s^2 (useActiveTCP=true) feature=Base
    Waypoint Waypoint_12: TCP in base x=-121.283 y=-195.081 z=269.514 mm, rx=-2.167 ry=2.2415 rz=-0.0076 rad; joints [-88.099, -64.133, -118.46, -88.049, 91.631, -85.899] deg
